% RSLogix 500 project Variador_remoto_3hilos.RSS, saved by version 8.30.00.16 %
PROJECT "UNTITLED"    % processor: Bul.1763 MicroLogix 1100 Series B %

PROGRAM FILES
  LAD 2   11 rungs

DATA FILES
  O0 OUTPUT  6 elements
  I1 INPUT  12 elements
  S2 STATUS  66 elements
  B3 BINARY  1 elements
  T4 TIMER  1 elements
  C5 COUNTER  1 elements
  R6 CONTROL  1 elements
  N7 INTEGER  3 elements
  F8 FLOAT  9 elements

LADDER 2
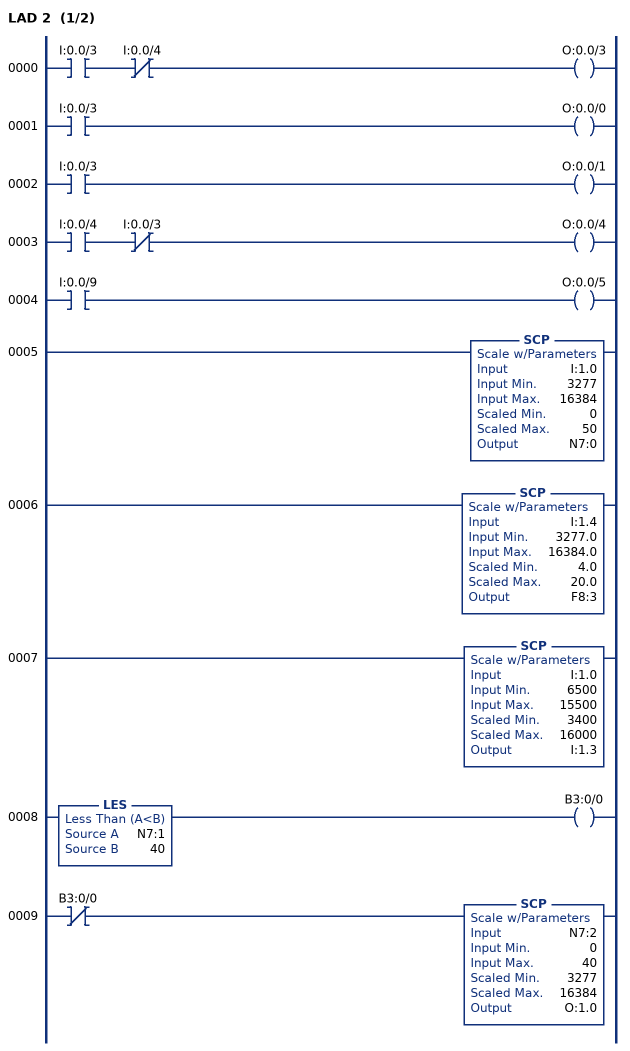
% Rung: 0 %
SOR XIC I:0.0/3 XIO I:0.0/4 OTE O:0.0/3 EOR
% Rung: 1 %
SOR XIC I:0.0/3 OTE O:0.0/0 EOR
% Rung: 2 %
SOR XIC I:0.0/3 OTE O:0.0/1 EOR
% Rung: 3 %
SOR XIC I:0.0/4 XIO I:0.0/3 OTE O:0.0/4 EOR
% Rung: 4 %
SOR XIC I:0.0/9 OTE O:0.0/5 EOR
% Rung: 5 %
SOR SCP I:1.0 3277 16384 0 50 N7:0 EOR
% Rung: 6 %
SOR SCP I:1.4 3277.0 16384.0 4.0 20.0 F8:3 EOR
% Rung: 7 %
SOR SCP I:1.0 6500 15500 3400 16000 I:1.3 EOR
% Rung: 8 %
SOR LES N7:1 40 OTE B3:0/0 EOR
% Rung: 9 %
SOR XIO B3:0/0 SCP N7:2 0 40 3277 16384 O:1.0 EOR

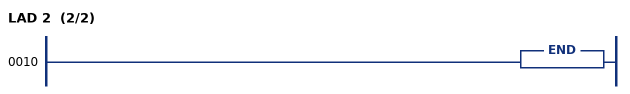
% Rung: 10 %
SOR END EOR

DATA TABLE (non-zero values as saved)
DATA N7
% N7:0 % 20 1 32
DATA F8
% F8:0 % 3 200 0.7003891 -0.0003051758 16384
